FUNCTION_BLOCK COMM_ADAPTER_SOCKET_PROXY_79152C3CB22C3086 (* Service Interface Function Block Type *)
  (* Standard: 61499-2 *)
  (* Version 0.0, 9/22/2017, bababen, nxtControl GmbH, template *)
  PACKAGE Main;
  (* Compiler Cpp nxtControl builtin 1.0 *)
  {SET_ATTRIBUTE(Configuration.GenericFBType.InterfaceParams, Runtime.System#<InterfaceList> <Sockets> <AdapterDeclaration Name="Out2" Type="BoolAdp" Namespace="Main" /> </Sockets> </InterfaceList>)}
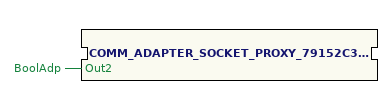
  SOCKETS
    Out2 : BoolAdp;
  END_SOCKETS
END_FUNCTION_BLOCK
